// TIA Portal V19 export
TYPE "LEXCHANGETRAY_typeNgConveyorEm_recieve_interface"
// stored: Access Published
   STRUCT
      handlingXyz { S7_SetPoint := 'True'} : "LEXCHANGETRAY_typeNgConveyorEm_toHandlingXyzRecieve";
   END_STRUCT;
END_TYPE
